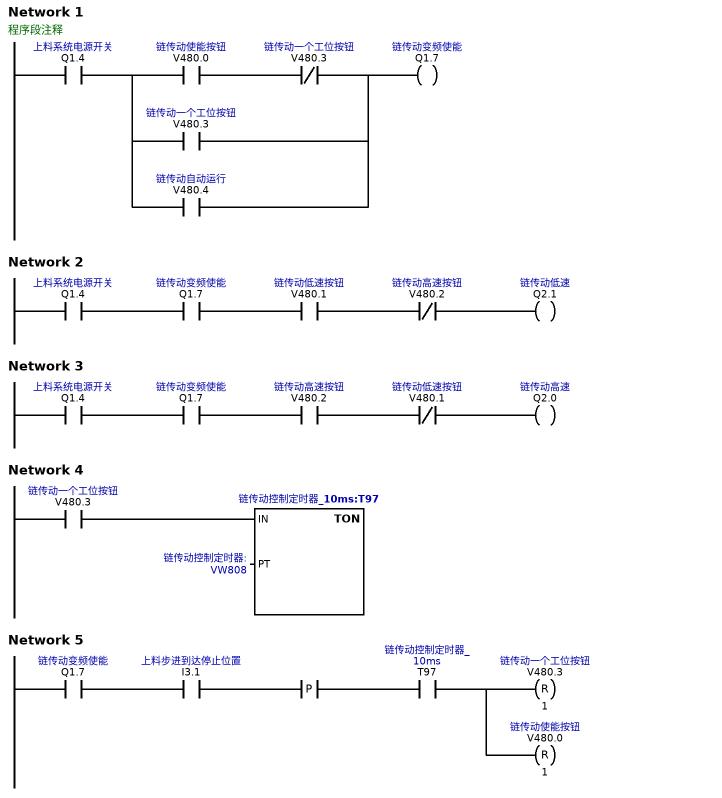
[picture p24: SBR19 networks 1-5]
Network 1
// 程序段注释
LD     上料系统电源开关:Q1.4
LD     链传动使能按钮:V480.0
AN     链传动一个工位按钮:V480.3
O      链传动一个工位按钮:V480.3
O      链传动自动运行:V480.4
ALD
=      链传动变频使能:Q1.7
Network 2
LD     上料系统电源开关:Q1.4
A      链传动变频使能:Q1.7
A      链传动低速按钮:V480.1
AN     链传动高速按钮:V480.2
=      链传动低速:Q2.1
Network 3
LD     上料系统电源开关:Q1.4
A      链传动变频使能:Q1.7
A      链传动高速按钮:V480.2
AN     链传动低速按钮:V480.1
=      链传动高速:Q2.0
Network 4
LD     链传动一个工位按钮:V480.3
TON    链传动控制定时器_10ms:T97, 链传动控制定时器:VW808
Network 5
LD     链传动变频使能:Q1.7
A      上料步进到达停止位置:I3.1
EU
A      链传动控制定时器_10ms:T97
R      链传动一个工位按钮:V480.3, 1
R      链传动使能按钮:V480.0, 1
END_SUBROUTINE_BLOCK

SUBROUTINE_BLOCK 数据初始化:SBR20
TITLE=子程序注释
BEGIN
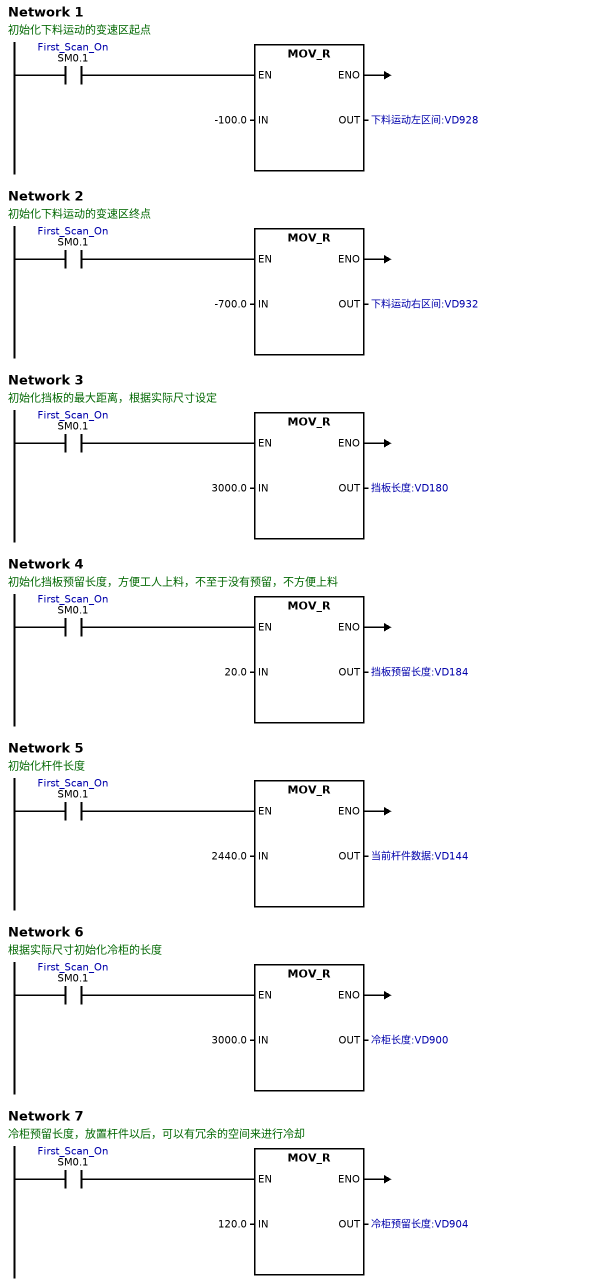
Network 1
// 初始化下料运动的变速区起点
LD     First_Scan_On:SM0.1
MOVR   -100.0, 下料运动左区间:VD928
Network 2
// 初始化下料运动的变速区终点
LD     First_Scan_On:SM0.1
MOVR   -700.0, 下料运动右区间:VD932
Network 3
// 初始化挡板的最大距离，根据实际尺寸设定
LD     First_Scan_On:SM0.1
MOVR   3000.0, 挡板长度:VD180
Network 4
// 初始化挡板预留长度，方便工人上料，不至于没有预留，不方便上料
LD     First_Scan_On:SM0.1
MOVR   20.0, 挡板预留长度:VD184
Network 5
// 初始化杆件长度
LD     First_Scan_On:SM0.1
MOVR   2440.0, 当前杆件数据:VD144
Network 6
// 根据实际尺寸初始化冷柜的长度
LD     First_Scan_On:SM0.1
MOVR   3000.0, 冷柜长度:VD900
Network 7
// 冷柜预留长度，放置杆件以后，可以有冗余的空间来进行冷却
LD     First_Scan_On:SM0.1
MOVR   120.0, 冷柜预留长度:VD904
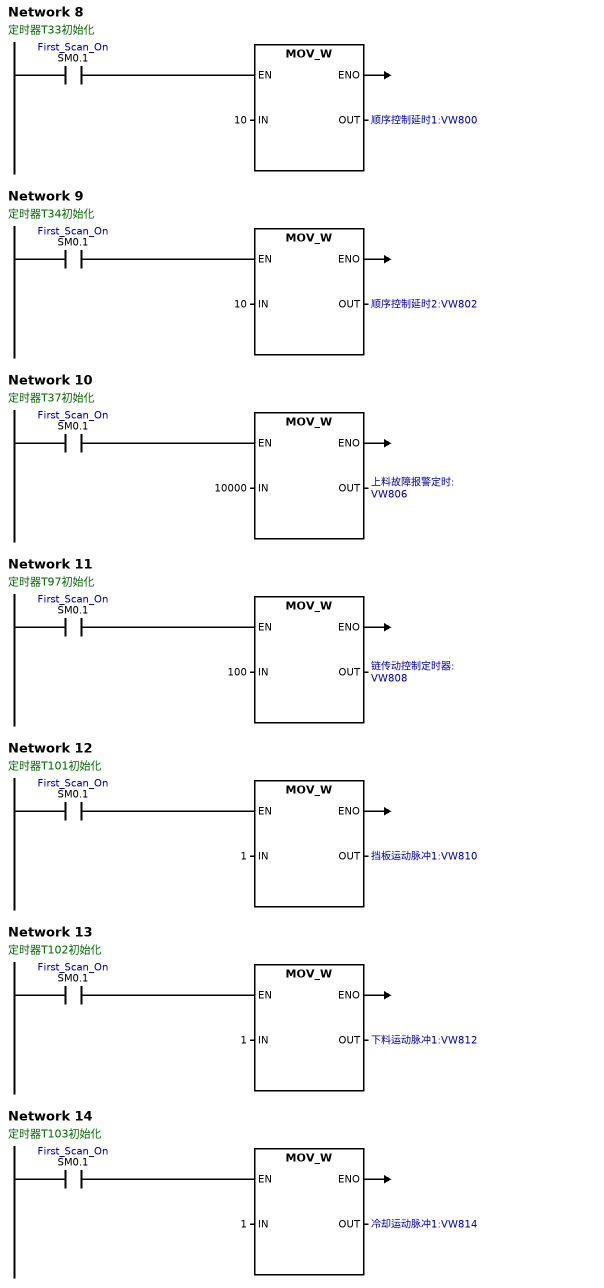
Network 8
// 定时器T33初始化
LD     First_Scan_On:SM0.1
MOVW   10, 顺序控制延时1:VW800
Network 9
// 定时器T34初始化
LD     First_Scan_On:SM0.1
MOVW   10, 顺序控制延时2:VW802
Network 10
// 定时器T37初始化
LD     First_Scan_On:SM0.1
MOVW   10000, 上料故障报警定时:VW806
Network 11
// 定时器T97初始化
LD     First_Scan_On:SM0.1
MOVW   100, 链传动控制定时器:VW808
Network 12
// 定时器T101初始化
LD     First_Scan_On:SM0.1
MOVW   1, 挡板运动脉冲1:VW810
Network 13
// 定时器T102初始化
LD     First_Scan_On:SM0.1
MOVW   1, 下料运动脉冲1:VW812
Network 14
// 定时器T103初始化
LD     First_Scan_On:SM0.1
MOVW   1, 冷却运动脉冲1:VW814
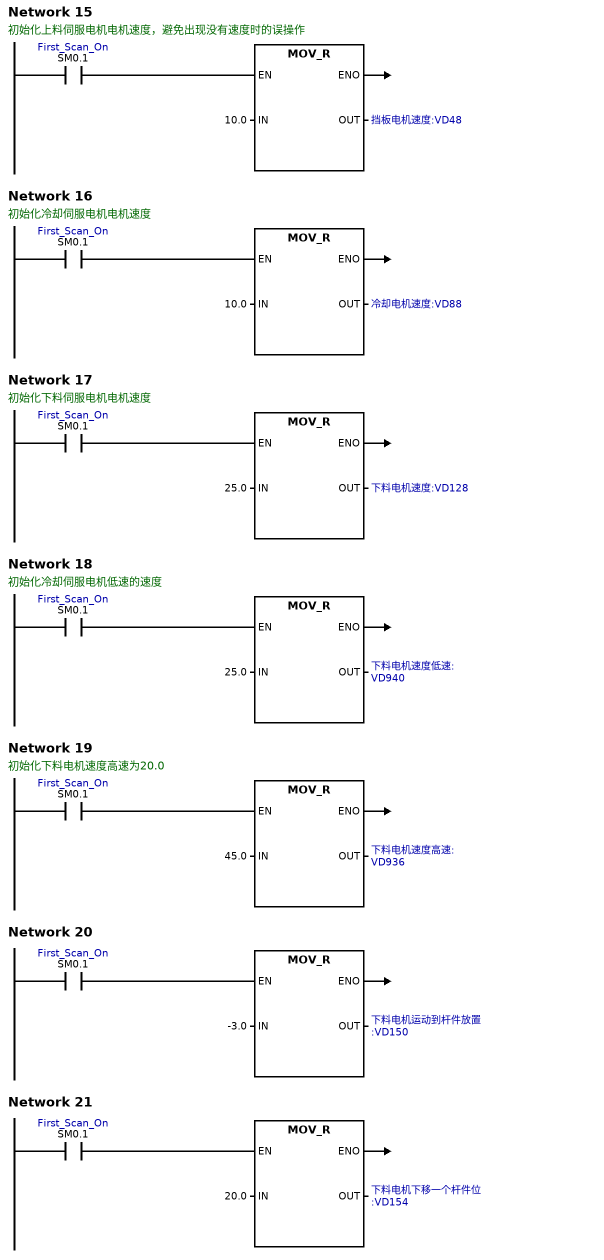
Network 15
// 初始化上料伺服电机电机速度，避免出现没有速度时的误操作
LD     First_Scan_On:SM0.1
MOVR   10.0, 挡板电机速度:VD48
Network 16
// 初始化冷却伺服电机电机速度
LD     First_Scan_On:SM0.1
MOVR   10.0, 冷却电机速度:VD88
Network 17
// 初始化下料伺服电机电机速度
LD     First_Scan_On:SM0.1
MOVR   25.0, 下料电机速度:VD128
Network 18
// 初始化冷却伺服电机低速的速度
LD     First_Scan_On:SM0.1
MOVR   25.0, 下料电机速度低速:VD940
Network 19
// 初始化下料电机速度高速为20.0
LD     First_Scan_On:SM0.1
MOVR   45.0, 下料电机速度高速:VD936
Network 20
LD     First_Scan_On:SM0.1
MOVR   -3.0, 下料电机运动到杆件放置:VD150
Network 21
LD     First_Scan_On:SM0.1
MOVR   20.0, 下料电机下移一个杆件位:VD154
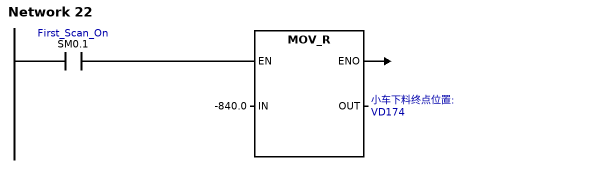
Network 22
LD     First_Scan_On:SM0.1
MOVR   -840.0, 小车下料终点位置:VD174
END_SUBROUTINE_BLOCK

SUBROUTINE_BLOCK 故障报警:SBR21
TITLE=子程序注释
BEGIN
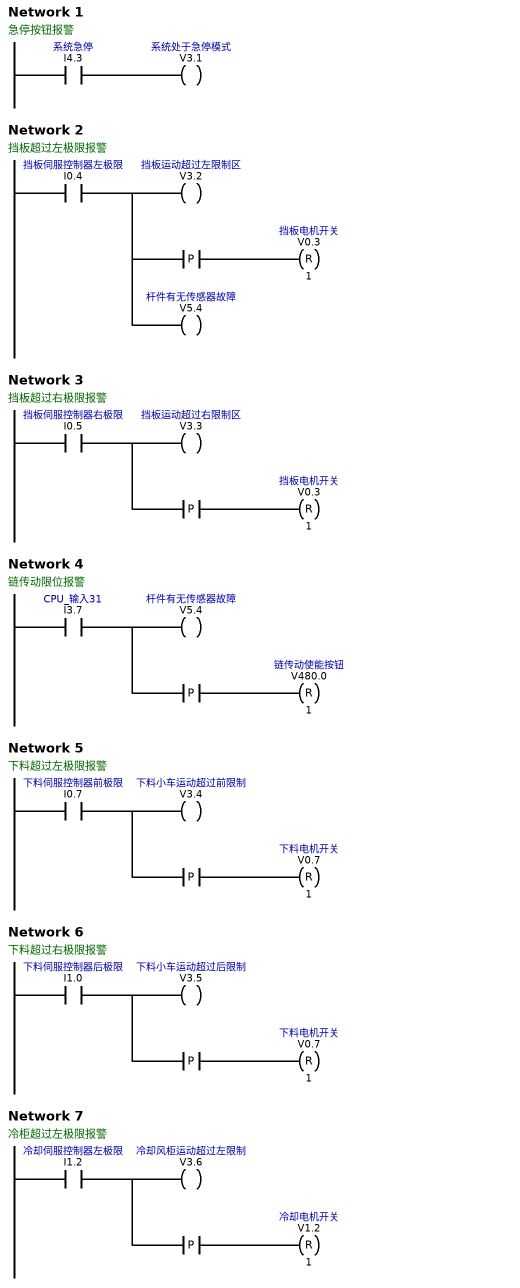
Network 1
// 急停按钮报警
LD     系统急停:I4.3
=      系统处于急停模式:V3.1
Network 2
// 挡板超过左极限报警
LD     挡板伺服控制器左极限:I0.4
LPS
=      挡板运动超过左限制区:V3.2
EU
R      挡板电机开关:V0.3, 1
LPP
=      杆件有无传感器故障:V5.4
Network 3
// 挡板超过右极限报警
LD     挡板伺服控制器右极限:I0.5
=      挡板运动超过右限制区:V3.3
EU
R      挡板电机开关:V0.3, 1
Network 4
// 链传动限位报警
LD     CPU_输入31:I3.7
=      杆件有无传感器故障:V5.4
EU
R      链传动使能按钮:V480.0, 1
Network 5
// 下料超过左极限报警
LD     下料伺服控制器前极限:I0.7
=      下料小车运动超过前限制:V3.4
EU
R      下料电机开关:V0.7, 1
Network 6
// 下料超过右极限报警
LD     下料伺服控制器后极限:I1.0
=      下料小车运动超过后限制:V3.5
EU
R      下料电机开关:V0.7, 1
Network 7
// 冷柜超过左极限报警
LD     冷却伺服控制器左极限:I1.2
=      冷却风柜运动超过左限制:V3.6
EU
R      冷却电机开关:V1.2, 1
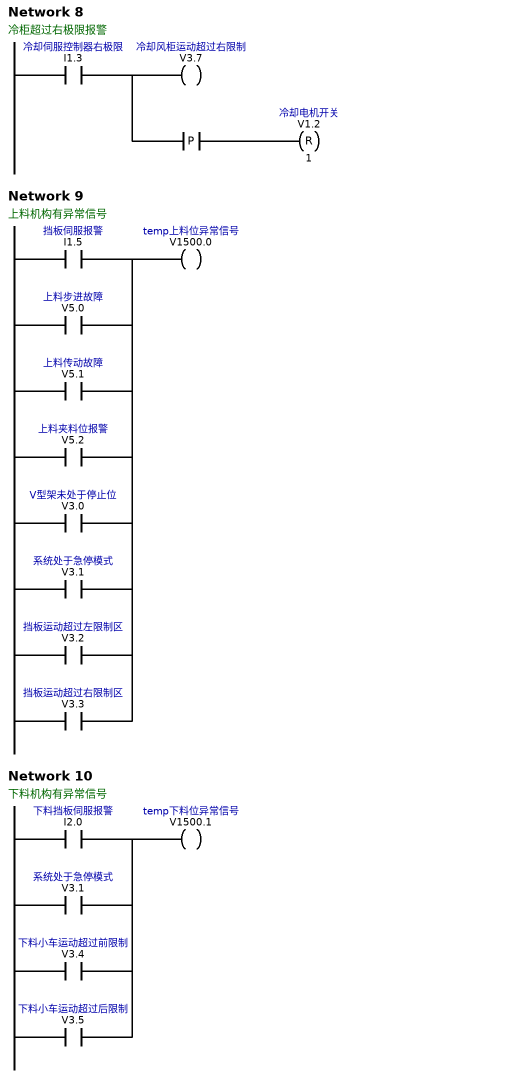
Network 8
// 冷柜超过右极限报警
LD     冷却伺服控制器右极限:I1.3
=      冷却风柜运动超过右限制:V3.7
EU
R      冷却电机开关:V1.2, 1
Network 9
// 上料机构有异常信号
LD     挡板伺服报警:I1.5
O      上料步进故障:V5.0
O      上料传动故障:V5.1
O      上料夹料位报警:V5.2
O      V型架未处于停止位:V3.0
O      系统处于急停模式:V3.1
O      挡板运动超过左限制区:V3.2
O      挡板运动超过右限制区:V3.3
=      temp上料位异常信号:V1500.0
Network 10
// 下料机构有异常信号
LD     下料挡板伺服报警:I2.0
O      系统处于急停模式:V3.1
O      下料小车运动超过前限制:V3.4
O      下料小车运动超过后限制:V3.5
=      temp下料位异常信号:V1500.1
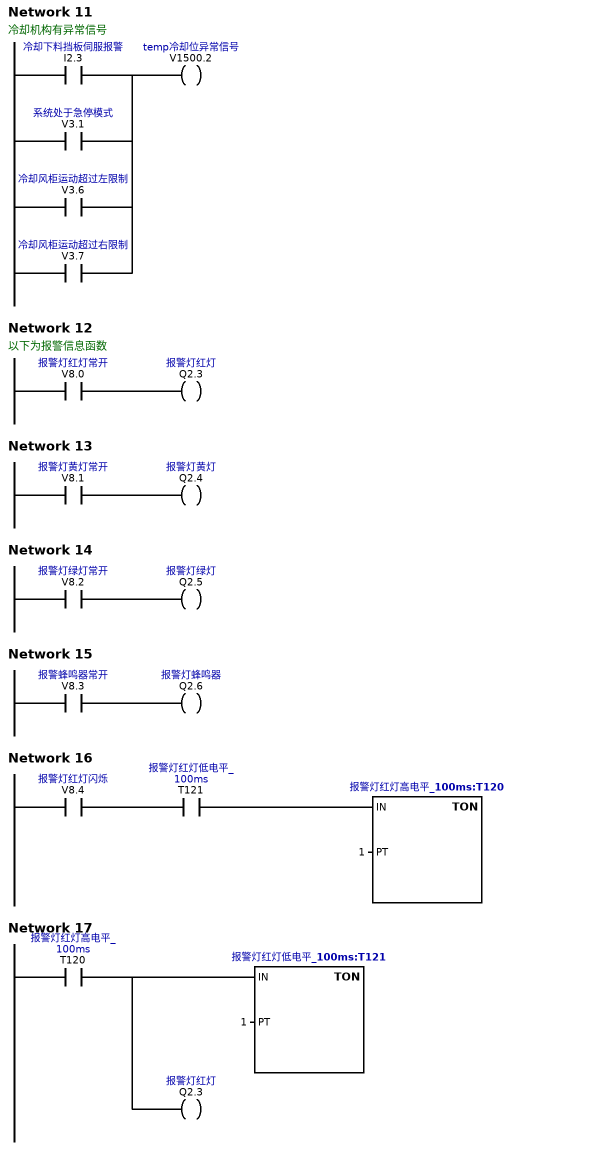
Network 11
// 冷却机构有异常信号
LD     冷却下料挡板伺服报警:I2.3
O      系统处于急停模式:V3.1
O      冷却风柜运动超过左限制:V3.6
O      冷却风柜运动超过右限制:V3.7
=      temp冷却位异常信号:V1500.2
Network 12
// 以下为报警信息函数
LD     报警灯红灯常开:V8.0
=      报警灯红灯:Q2.3
Network 13
LD     报警灯黄灯常开:V8.1
=      报警灯黄灯:Q2.4
Network 14
LD     报警灯绿灯常开:V8.2
=      报警灯绿灯:Q2.5
Network 15
LD     报警蜂鸣器常开:V8.3
=      报警灯蜂鸣器:Q2.6
Network 16
LD     报警灯红灯闪烁:V8.4
A      报警灯红灯低电平_100ms:T121
TON    报警灯红灯高电平_100ms:T120, 1
Network 17
LD     报警灯红灯高电平_100ms:T120
TON    报警灯红灯低电平_100ms:T121, 1
=      报警灯红灯:Q2.3
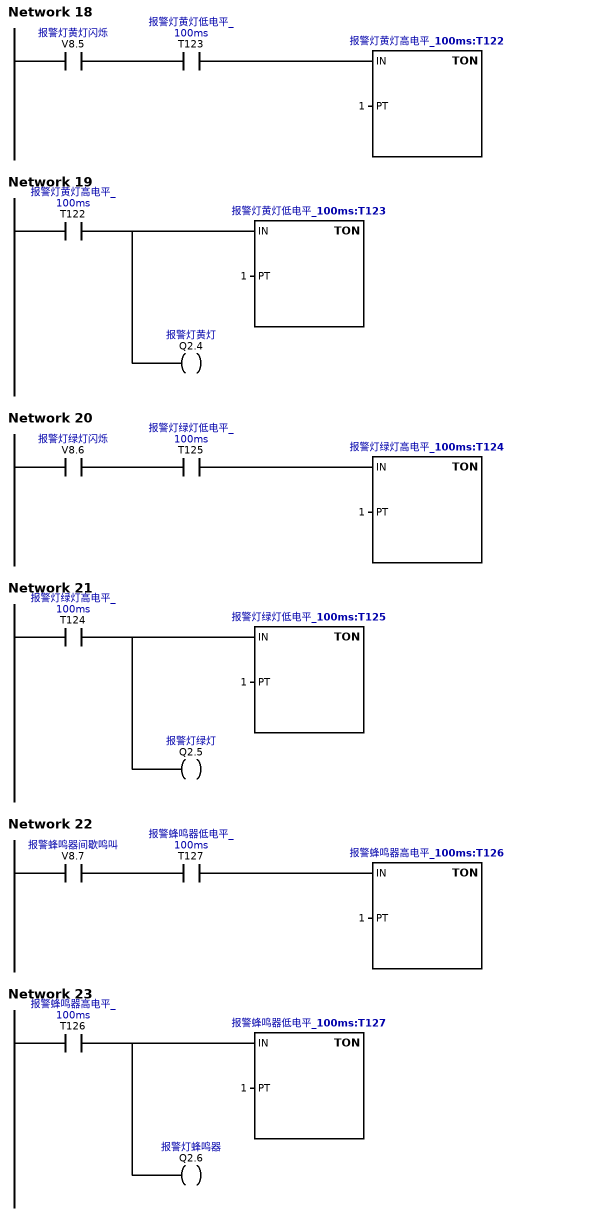
Network 18
LD     报警灯黄灯闪烁:V8.5
A      报警灯黄灯低电平_100ms:T123
TON    报警灯黄灯高电平_100ms:T122, 1
Network 19
LD     报警灯黄灯高电平_100ms:T122
TON    报警灯黄灯低电平_100ms:T123, 1
=      报警灯黄灯:Q2.4
Network 20
LD     报警灯绿灯闪烁:V8.6
A      报警灯绿灯低电平_100ms:T125
TON    报警灯绿灯高电平_100ms:T124, 1
Network 21
LD     报警灯绿灯高电平_100ms:T124
TON    报警灯绿灯低电平_100ms:T125, 1
=      报警灯绿灯:Q2.5
Network 22
LD     报警蜂鸣器间歇鸣叫:V8.7
A      报警蜂鸣器低电平_100ms:T127
TON    报警蜂鸣器高电平_100ms:T126, 1
Network 23
LD     报警蜂鸣器高电平_100ms:T126
TON    报警蜂鸣器低电平_100ms:T127, 1
=      报警灯蜂鸣器:Q2.6
END_SUBROUTINE_BLOCK
